KUKA KRL data list: PolishReplaceHead.dat

&ACCESS RVO
&REL 79
&COMMENT Polish Replace Head 250608
defdat PolishReplaceHead

decl state_t State
decl int Offset = 0
decl char Msg[128]

enddat
